INTERFACE ITF_XtsMoverAxis

PROPERTY Acceleration : mc_lreal
GET
END_GET
SET
END_SET
END_PROPERTY

METHOD ActivateTrack : HRESULT
VAR_INPUT
	NewTrack : OTCID;
	Track : I_XtsTrack;
END_VAR
END_METHOD

PROPERTY AxisRef : Reference to Axis_ref
GET
END_GET
END_PROPERTY

PROPERTY Deceleration : mc_lreal
GET
END_GET
SET
END_SET
END_PROPERTY

METHOD DisableMover : HRESULT
VAR_INPUT
END_VAR
END_METHOD

METHOD EnableMover : HRESULT
VAR_INPUT
END_VAR
END_METHOD

PROPERTY Gap : MC_LREAL
GET
END_GET
SET
END_SET
END_PROPERTY

METHOD PUBLIC Gear : HRESULT
VAR_INPUT
	MasterPosition : MC_LREAL;
	SlavePosition : MC_LREAL;
END_VAR
END_METHOD

METHOD HaltAxis : HRESULT
VAR_INPUT
END_VAR
END_METHOD

PROPERTY PUBLIC IdentInGroup : IDENT_IN_GROUP_REF
GET
END_GET
END_PROPERTY

METHOD isMoverAtPosition : BOOL
VAR_INPUT
	Position : MC_LREAL;
END_VAR
END_METHOD

METHOD isMoverDetected : BOOL
VAR_INPUT
END_VAR
END_METHOD

METHOD isMoverEnabled : BOOL
VAR_INPUT
END_VAR
END_METHOD

METHOD isMoverStationary : BOOL
VAR_INPUT
END_VAR
END_METHOD

PROPERTY Jerk : mc_lreal
GET
END_GET
SET
END_SET
END_PROPERTY

PROPERTY PUBLIC MoverErrorID : DWORD
GET
END_GET
END_PROPERTY

PROPERTY PUBLIC MoversActiveTrack : OTCID
GET
END_GET
END_PROPERTY

PROPERTY PUBLIC MoverXtsIoEnvInterface : I_TcIoXtsXpuMover
GET
END_GET
SET
END_SET
END_PROPERTY

METHOD MoveTo : HRESULT
VAR_INPUT
	RequiredPosition : MC_LREAL;
	MoveVelocity : MC_LREAL;
	NonModuloMove : BOOL;
END_VAR
END_METHOD

PROPERTY MyCAGroup : ITF_CAMover
GET
END_GET
SET
END_SET
END_PROPERTY

PROPERTY MyMasterRef : REFERENCE TO AXIS_REF
GET
END_GET
SET
END_SET
END_PROPERTY

PROPERTY PositiveDirectionOnly : BOOL
GET
END_GET
SET
END_SET
END_PROPERTY

METHOD ResetAxis : HRESULT
VAR_INPUT
END_VAR
END_METHOD

METHOD TriggerMoverArrive : BOOL
VAR_INPUT
END_VAR
END_METHOD

METHOD TriggerMoverLeave : BOOL
VAR_INPUT
END_VAR
END_METHOD

END_INTERFACE

(* stored: Version 1.1.0.1, ProductVersion 3.1.4026.11
   Itf ITF_XtsMoverAxis: Id {3dcfc709-5ede-408c-bb46-9ff1ab7ba3a2}
   Folder Administration: Id {4954b02a-5467-474b-b4cc-9e953c27295d}
   Folder Commands: Id {106fb726-2896-4a76-8d42-ca08d03a1871}
   Folder Dynamics: Id {f06c35fd-2445-4fb9-97b8-caf92ac08b38}
   Folder Status: Id {6f079834-b92a-4de6-abe6-7b90d541a1af}
   Property Acceleration: Id {968dd06c-5bd7-474e-8a7d-3c6c7a848d78}
   Get Get: Id {ad3ccb1b-ebe0-4c79-851d-54fe9678941a}
   Set Set: Id {ad0cd55c-ffe5-41e5-89e5-44c936340625}
   Method ActivateTrack: Id {ba6e327e-25a9-4189-a1a0-64429eeca8b6}
   Property AxisRef: Id {b9459322-2642-4758-9d1a-f140abbed4b3}
   Get Get: Id {fca9e840-ce68-48f6-aaf7-b30da4df166b}
   Property Deceleration: Id {925224a3-633f-4afb-a6bb-5e2282bf0166}
   Get Get: Id {ee77943b-5dd1-4851-bfac-c1f6c08f427a}
   Set Set: Id {cf0b19b4-9657-4139-bc2e-afb49fbc4d88}
   Method DisableMover: Id {ab15092e-3fa3-489a-9dc6-5a5b357cf3f5}
   Method EnableMover: Id {12e4840c-ab85-431d-8aa9-ce712b4847e4}
   Property Gap: Id {fb9a5121-dbab-42c7-b05b-e0e4367182c8}
   Get Get: Id {0b18224e-8e16-4474-96e3-0906bc0c9a81}
   Set Set: Id {2dea6ad0-842c-4a1e-91cb-fd845bae918b}
   Method Gear: Id {e0c78185-a7ab-4223-b289-235f40f7bfac}
   Method HaltAxis: Id {881642ff-213b-4030-944f-bd624c008c64}
   Property IdentInGroup: Id {892b953d-abf1-49a8-bf89-421385c1791d}
   Get Get: Id {b023befb-8f40-468b-ada4-daaf368f7d24}
   Method isMoverAtPosition: Id {bc703c47-0b4d-4374-b07c-1240b49b484e}
   Method isMoverDetected: Id {bebf9077-4fa3-41f0-a58b-68e771a6d3a7}
   Method isMoverEnabled: Id {2ad921d2-fe23-4c3a-8e9a-22becef3f18a}
   Method isMoverStationary: Id {7e7da463-610e-4ddb-b6e7-ef0925f02451}
   Property Jerk: Id {8063437d-ace9-4769-bdaf-bbbe2e6cdcb8}
   Get Get: Id {7a71a7bc-503a-407e-bd5c-807dc27f8a07}
   Set Set: Id {943274ff-ff90-4228-a079-22863adf0d58}
   Property MoverErrorID: Id {b22f6e77-1f1b-46fd-9beb-24cd7598be7b}
   Get Get: Id {a8d82d04-fa66-4bdd-839c-2ee85269a247}
   Property MoversActiveTrack: Id {f033ba71-1699-4f66-8762-38178a524724}
   Get Get: Id {ab30b8a7-22d3-4a5c-a941-ce17b5400c54}
   Property MoverXtsIoEnvInterface: Id {192fc175-f0e7-4171-9425-47deb3799f9d}
   Get Get: Id {e7a8a250-ae9b-4ad7-bf97-7690d04cb985}
   Set Set: Id {f163ce07-1471-4036-baf2-4d783308d9bd}
   Method MoveTo: Id {ff1a94f0-d91e-4f1f-8540-ce9d25779d5e}
   Property MyCAGroup: Id {7bdbd73e-c8bd-4342-9139-b02fb8b34afa}
   Get Get: Id {02d1886c-e164-4472-af91-ae6725f23e23}
   Set Set: Id {0add7ecc-1e34-4c45-86ea-05d00a10668e}
   Property MyMasterRef: Id {ef955fbf-3876-4064-a941-698a35c297a1}
   Get Get: Id {a4aadfe1-030c-4097-bbb9-7ab611ed666a}
   Set Set: Id {f70f72b0-a05b-4221-b76a-6ab9157d064d}
   Property PositiveDirectionOnly: Id {ed0ab13d-fd6f-4b8b-a5b2-30d977b85665}
   Get Get: Id {ca7928e2-abd0-4257-bca9-4dcae3e4cfec}
   Set Set: Id {89d703fe-11d9-4067-a762-3ca15c65b604}
   Method ResetAxis: Id {6858a2d4-c501-4639-b0f6-64db9416c8f9}
   Method TriggerMoverArrive: Id {ce200a85-cca0-47d0-8b7e-22e3d01f8c11}
   Method TriggerMoverLeave: Id {fe2ebe40-b0b7-4184-8656-d9f18bf6a0ec} *)
